FUNCTION_BLOCK FB_PressureTransducer EXTENDS FB_Device
VAR_INPUT
	nSensorPressure: INT; //Pressure analog input
	nSensorTemperature:INT;//Temperature analog input 
	st_AnalogPressureTempdata:ST_AnalogPressureTemp;//Configuration struct 
	sTag : T_MaxString;
END_VAR
VAR_OUTPUT
	rEngPressure:REAL;//Pressure in BAR.
	rEngTemperature:REAL;//Temperature in Degrees C.
END_VAR

M_CyclicLogic();

METHOD M_CyclicLogic : HRESULT
VAR
	rNormPressure:REAL;
	rNormTemperature:REAL;
END_VAR
//Call M_CyclicLogic from FB_Device 
hr:=SUPER^.M_CyclicLogic();
IF bDeviceEnable THEN
	//Normalise the analog inputs 
   rNormPressure    := (INT_TO_REAL(nSensorPressure)    - INT_TO_REAL(st_AnalogPressureTempdata.nRawMin)) / (INT_TO_REAL(st_AnalogPressureTempdata.nRawMax) - INT_TO_REAL(st_AnalogPressureTempdata.nRawMin));
   rNormTemperature := (INT_TO_REAL(nSensorTemperature) - INT_TO_REAL(st_AnalogPressureTempdata.nRawMin)) / (INT_TO_REAL(st_AnalogPressureTempdata.nRawMax) - INT_TO_REAL(st_AnalogPressureTempdata.nRawMin));
   
   //Scale analog inputs to the Engineering process values, using config struct parameters
   rEngPressure:=st_AnalogPressureTempdata.rPressureMinSP + rNormPressure * (st_AnalogPressureTempdata.rPressureMaxSP - st_AnalogPressureTempdata.rPressureMinSP);
   rEngTemperature:=st_AnalogPressureTempdata.rTemperatureMinSP + rNormTemperature * (st_AnalogPressureTempdata.rTemperatureMaxSP - st_AnalogPressureTempdata.rTemperatureMinSP);
END_IF

//Evaluate pressure state 
M_PressureState();
END_METHOD

METHOD M_PressureState : BOOL
//Evaluate pressure value against warning and error values.
IF (rEngPressure > st_AnalogPressureTempdata.rWarninglevel) AND (rEngPressure < st_AnalogPressureTempdata.rErrorLevel) THEN
	bWarning:=TRUE;
ELSIF rEngPressure > st_AnalogPressureTempdata.rErrorLevel THEN
	bError:=TRUE;
ELSE 
	bWarning:=FALSE;
END_IF
END_METHOD

END_FUNCTION_BLOCK

(* stored: Version 1.1.0.1
   POU FB_PressureTransducer: Id {4a351574-9fd7-451d-b391-c9b46c5a302c}, SpecialFunc None
   Method M_CyclicLogic: Id {1ef18ec2-39ea-4a7a-9812-158fef41a970}
   Method M_PressureState: Id {5a80939a-4228-4bfa-a79b-b4ef01743c70} *)
